{attribute 'linkalways'} 
{attribute 'no_explicit_call' := 'This FB is a CLASS and must be accessed using methods or properties'}
{attribute 'enable_dynamic_creation'}
FUNCTION_BLOCK _ETcVnInitializableFunction EXTENDS EnumDatatypeBase
VAR
	localData : ETcVnInitializableFunction;
	activeData : REFERENCE TO ETcVnInitializableFunction;
	enumBaseDatatype : _DINT(localData);
END_VAR

METHOD PRIVATE AddLocalEnumeration
VAR_INPUT
	Enumeration : T_MAXSTRING;
	Value : ETcVnInitializableFunction;
END_VAR
AddEnumeration(Enumeration, Value);
END_METHOD

PROPERTY PUBLIC Address : PVOID
GET
Address := ADR(activeData);
END_GET
END_PROPERTY

METHOD PUBLIC ClearReference
VAR_INPUT
END_VAR
activeData REF= localData;
SetBaseDatatypeReference();
END_METHOD

METHOD PUBLIC Clone : I_Datatype
VAR
    pClone : POINTER TO _ETcVnInitializableFunction;
END_VAR
pClone := __NEW(_ETcVnInitializableFunction(InitialValue := Value));
Clone := pClone^;
END_METHOD

METHOD FB_init : BOOL
VAR_INPUT
	bInitRetains : BOOL; // if TRUE, the retain variables are initialized (warm start / cold start)
	bInCopyCode : BOOL;  // if TRUE, the instance afterwards gets moved into the copy code (online change)
	InitialValue : ETcVnInitializableFunction;
END_VAR
localData := InitialValue;
AddBaseDatatype(enumBaseDatatype);
ClearReference();

AddLocalEnumeration('TCVN_IF_OCR', ETcVnInitializableFunction.TCVN_IF_OCR);
END_METHOD

PROPERTY PUBLIC Identifier : T_MAXSTRING
GET
Identifier := 'ETcVnInitializableFunction';
END_GET
END_PROPERTY

METHOD IsEnumeratorValueEqual : BOOL
VAR_INPUT
	Enumerator : I_KeyValueForwardEnumerator;
END_VAR
VAR
	storedValue : ETcVnInitializableFunction;
END_VAR
IF NOT Enumerator.TryGet(storedValue) THEN
	RETURN;
END_IF

IsEnumeratorValueEqual := storedValue = activeData;
END_METHOD

METHOD PUBLIC MakeReferenceTo
VAR_INPUT
	ReferenceTarget : REFERENCE TO ETcVnInitializableFunction;
END_VAR
activeData REF= ReferenceTarget;
SetBaseDatatypeReference();
END_METHOD

METHOD PROTECTED SetBaseDatatypeReference
VAR_INPUT
END_VAR
enumBaseDatatype.MakeReferenceTo(activeData);
END_METHOD

PROPERTY PUBLIC Size : UDINT
GET
Size := SIZEOF(activeData);
END_GET
END_PROPERTY

METHOD TryMakeReferenceTo : BOOL
VAR_INPUT
	Target : I_Datatype;
END_VAR
VAR
	targetAsEnum : I_EnumDatatype;
	pTargetData : POINTER TO ETcVnInitializableFunction;
END_VAR
IF NOT Target.TryResolveAsEnumDatatype(targetAsEnum) THEN
	RETURN;
END_IF

IF targetAsEnum.Identifier <> Identifier THEN
	RETURN;
END_IF

pTargetData := Target.Address;
activeData REF= pTargetData^;
SetBaseDatatypeReference();
TryMakeReferenceTo := TRUE;
END_METHOD

PROPERTY PUBLIC Value : ETcVnInitializableFunction
GET
Value := activeData;
END_GET
SET
activeData := Value;
END_SET
END_PROPERTY

END_FUNCTION_BLOCK

(* stored: Version 1.1.0.1, ProductVersion 3.1.4024.12
   POU _ETcVnInitializableFunction: Id {862eef73-5f14-4f78-a11c-c75864defc75}, SpecialFunc None
   Folder Constructor: Id {62dfc604-e947-44ad-a8e1-65f7a999be8c}
   Folder Private: Id {df443a66-f46e-4018-851b-8ef7308bed76}
   Folder Protected: Id {3bdd63e4-73ac-4665-b59b-994a4adb1975}
   Method AddLocalEnumeration: Id {04a5cd4a-267b-4df7-9248-06a05530debf}
   Property Address: Id {1e90302e-9020-4684-bbb0-cebe3761fb47}
   Get Get: Id {721a9ff9-f6a5-4537-8711-96bd0c8cc3ea}
   Method ClearReference: Id {2ac0d2b6-3575-4d6c-9a7a-dbfda221199b}
   Method Clone: Id {62de4d58-fca6-48e0-8c48-8ab3b5cd0095}
   Method FB_init: Id {8cfa8804-04a1-4df3-9bd0-ca7d29bfcb44}
   Property Identifier: Id {9be325f0-a991-402a-b043-aa9d837e8e78}
   Get Get: Id {d2f6e6bb-f81b-42dc-b736-002c61e603ed}
   Method IsEnumeratorValueEqual: Id {7ffb2227-f974-4111-aef8-333d8af11025}
   Method MakeReferenceTo: Id {a7329d25-d17a-4c19-9c6a-7385e05366bb}
   Method SetBaseDatatypeReference: Id {984a9145-35c9-492f-a7cc-ab2ba7c1d5ef}
   Property Size: Id {7d597dbf-10de-438d-ad43-7339306ed2ea}
   Get Get: Id {1eb1fda5-00fe-4a9f-adae-aed023cf5c65}
   Method TryMakeReferenceTo: Id {351a53f1-1e7b-4cc3-9591-184c7be8be7b}
   Property Value: Id {5b4bd8c3-b7d3-4c2f-a2b1-c6369314e516}
   Get Get: Id {43d54c80-2472-4184-b9aa-b63e7944e156}
   Set Set: Id {0043eb86-7349-45f4-8e0e-7877c6167ae0} *)
